% RSLogix 500 project PLC Runtime Tracker with Hour Meter.RSS, saved by version 8.30.00.16 %
PROJECT "UNTITLED"    % processor: Bul.1763 MicroLogix 1100 Series B %

PROGRAM FILES
  LAD 2   9 rungs

DATA FILES
  O0 OUTPUT  4 elements
  I1 INPUT  6 elements
  S2 STATUS  66 elements
  B3 BINARY  1 elements
  T4 TIMER  1 elements
  C5 COUNTER  4 elements
  R6 CONTROL  1 elements
  N7 INTEGER  4 elements
  F8 FLOAT  1 elements

LADDER 2
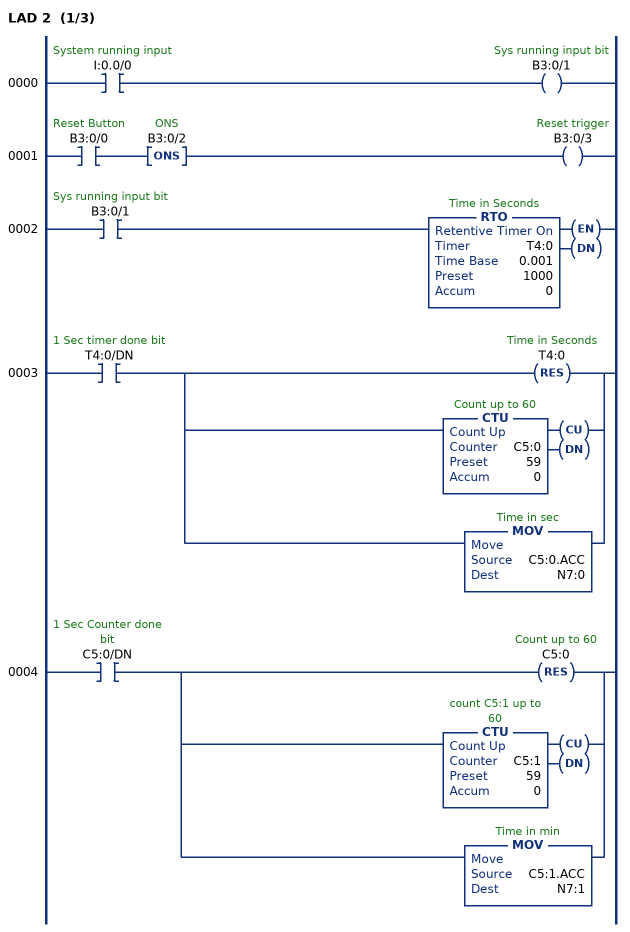
% Rung: 0 %
SOR XIC I:0.0/0 OTE B3:0/1 EOR
%   I:0.0/0  "System running input" %
%   B3:0/1  "Sys running input bit" %
% Rung: 1 %
SOR XIC B3:0/0 ONS B3:0/2 OTE B3:0/3 EOR
%   B3:0/0  "Reset Button" %
%   B3:0/2  "ONS" %
%   B3:0/3  "Reset trigger" %
% Rung: 2 %
SOR XIC B3:0/1 RTO T4:0 0.001 1000 0 EOR
%   B3:0/1  "Sys running input bit" %
%   T4:0  "Time in Seconds" %
% Rung: 3 %
SOR XIC T4:0/DN BST RES T4:0 NXB CTU C5:0 59 0 NXB MOV C5:0.ACC N7:0 BND EOR
%   T4:0/DN  "1 Sec timer done bit" %
%   T4:0  "Time in Seconds" %
%   C5:0  "Count up to 60" %
%   N7:0  "Time in sec" %
% Rung: 4 %
SOR XIC C5:0/DN BST RES C5:0 NXB CTU C5:1 59 0 NXB MOV C5:1.ACC N7:1 BND EOR
%   C5:0/DN  "1 Sec Counter done bit" %
%   C5:0  "Count up to 60" %
%   C5:1  "count C5:1 up to 60" %
%   N7:1  "Time in min" %

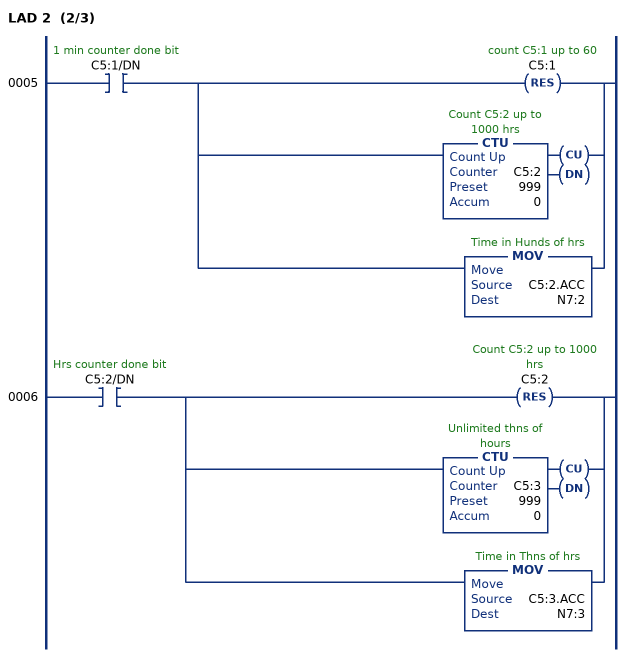
% Rung: 5 %
SOR XIC C5:1/DN BST RES C5:1 NXB CTU C5:2 999 0 NXB MOV C5:2.ACC N7:2 BND EOR
%   C5:1/DN  "1 min counter done bit" %
%   C5:1  "count C5:1 up to 60" %
%   C5:2  "Count C5:2 up to 1000 hrs" %
%   N7:2  "Time in Hunds of hrs" %
% Rung: 6 %
SOR XIC C5:2/DN BST RES C5:2 NXB CTU C5:3 999 0 NXB MOV C5:3.ACC N7:3 BND EOR
%   C5:2/DN  "Hrs counter done bit" %
%   C5:2  "Count C5:2 up to 1000 hrs" %
%   C5:3  "Unlimited thns of hours" %
%   N7:3  "Time in Thns of hrs" %

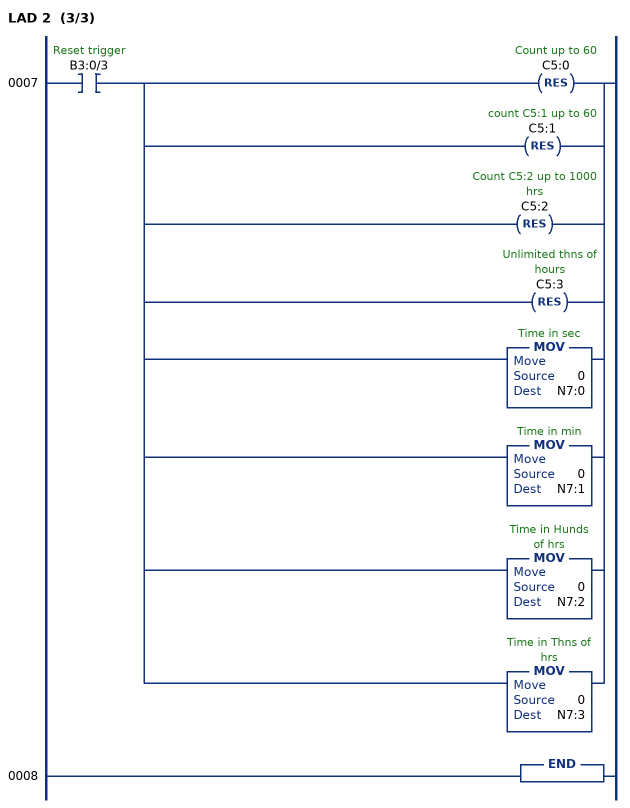
% Rung: 7 %
SOR XIC B3:0/3 BST RES C5:0 NXB RES C5:1 NXB RES C5:2 NXB RES C5:3 NXB MOV 0 N7:0 NXB MOV 0 N7:1 NXB MOV 0 N7:2 NXB MOV 0 N7:3 BND EOR
%   B3:0/3  "Reset trigger" %
%   C5:0  "Count up to 60" %
%   C5:1  "count C5:1 up to 60" %
%   C5:2  "Count C5:2 up to 1000 hrs" %
%   C5:3  "Unlimited thns of hours" %
%   N7:0  "Time in sec" %
%   N7:1  "Time in min" %
%   N7:2  "Time in Hunds of hrs" %
%   N7:3  "Time in Thns of hrs" %
% Rung: 8 %
SOR END EOR

DATA TABLE (non-zero values as saved)
DATA T4
% .PRE .ACC %
% T4:0 % 1000 0
DATA C5
% .PRE .ACC %
% C5:0 % 59 0
% C5:1 % 59 0
% C5:2 % 999 0
% C5:3 % 999 0
